FUNCTION TryConvert_REAL_TO_LREAL : BOOL
VAR_INPUT
	in : REAL;
	out : REFERENCE TO LREAL;
END_VAR

out := REAL_TO_LREAL(in);
TryConvert_REAL_TO_LREAL := TRUE;

END_FUNCTION

(* stored: Version 1.1.0.1, ProductVersion 3.1.4024.12
   POU TryConvert_REAL_TO_LREAL: Id {f5489566-6f99-4366-8639-dfc8e54832b5}, SpecialFunc None *)
